{attribute 'GeneratedUsingTerminal: EK1122-0000-0018'}
{attribute addProperty BoxType "EK1122-0000-0018"}
{attribute addProperty Id "Beckhoff_CXxxxxsub_EK1100EK1100_AB5A94672A_0001_CX1100_0004_0000CX1100_AB5A94672A_0003_CX1100_0004_0002CX1100_AB5A94672A_0004_CX5010_EtherCAT_slaveCX5010_EtherCAT_slave_08881C8E20A_0005_CX5010_EtherCAT_slaveCX5010_EtherCAT_slave_08881C8E20A_0006_CX5020_EtherCAT_slaveCX5020_EtherCAT_slave_08881C8E20A_0007_CX5020_EtherCAT_slaveCX5020_EtherCAT_slave_08881C8E20A_0008_CX8010_EtherCAT_slaveCX8010_EtherCAT_slave_08881C8E20A_0009_CX8010_EtherCAT_slaveCX8010_EtherCAT_slave_08881C8E20A_0010_CX8110_EtherCAT_slaveCX8110_EtherCAT_slave_08881C8E20A_0011_CX2020_EtherCAT_slaveCX2020_EtherCAT_slave_08881C8E20A_0012_CX2020_EtherCAT_slaveCX2020_EtherCAT_slave_08881C8E20A_0013_CX2020_EtherCAT_slaveCX2020_EtherCAT_slave_08881C8E20A_0014_CX2030_EtherCAT_slaveCX2030_EtherCAT_slave_08881C8E20A_0015_CX2030_EtherCAT_slaveCX2030_EtherCAT_slave_08881C8E20A_0016_CX2030_EtherCAT_slaveCX2030_EtherCAT_slave_08881C8E20A_0017_CX2033_EtherCAT_slaveCX2033_EtherCAT_slave_08881C8E20A_0018_CX2040_EtherCAT_slaveCX2040_EtherCAT_slave_08881C8E20A_0019_CX2040_EtherCAT_slaveCX2040_EtherCAT_slave_08881C8E20A_0020_CX2040_EtherCAT_slaveCX2040_EtherCAT_slave_08881C8E20A_0021_CX2042_EtherCAT_slaveCX2042_EtherCAT_slave_08881C8E20A_0022_CX2043_EtherCAT_slaveCX2043_EtherCAT_slave_08881C8E20A_0023_CX2062_EtherCAT_slaveCX2062_EtherCAT_slave_08881C8E20A_0024_CX2072_EtherCAT_slaveCX2072_EtherCAT_slave_08881C8E20A_0025_CX9020_EtherCAT_slaveCX9020_EtherCAT_slave_08881C8E20A_0026_CX9020_EtherCAT_slaveCX9020_EtherCAT_slave_08881C8E20A_0027_CX5120_EtherCAT_slaveCX5120_EtherCAT_slave_08881C8E20A_0028_CX5130_EtherCAT_slaveCX5130_EtherCAT_slave_08881C8E20A_0029_CX5140_EtherCAT_slaveCX5140_EtherCAT_slave_08881C8E20A_0030_CX5230_EtherCAT_slaveCX5230_EtherCAT_slave_08881C8E20A_0031_CX5240_EtherCAT_slaveCX5240_EtherCAT_slave_08881C8E20A_0002_CX1100_0004_0001CX1100_AB5A94672"}
{attribute addProperty CRC "3494610126"}
{attribute addProperty Size "568"}
TYPE Beckhoff_CXxxxxEK1122_D04B84CE EXTENDS EK1122_AB5A9467 :
STRUCT
	{attribute addProperty Name "Beckhoff_CXxxxxsub_EK1100"}
	{attribute addProperty PreviousPort "Beckhoff CXxxxxEK1122 : D"}
	Beckhoff_CXxxxxsub_EK1100 : EK1100_AB5A9467;
	{attribute addProperty Name "A_0001_CX1100_0004_0000"}
	{attribute addProperty PreviousPort "Beckhoff CXxxxxsub EK1100 : C"}
	A_0001_CX1100_0004_0000 : CX1100_AB5A9467;
	{attribute addProperty Name "A_0003_CX1100_0004_0002"}
	{attribute addProperty PreviousPort "A_0001(CX1100-0004-0000) : C"}
	A_0003_CX1100_0004_0002 : CX1100_AB5A9467;
	{attribute addProperty Name "A_0004_CX5010_EtherCAT_slave"}
	{attribute addProperty PreviousPort "Beckhoff CXxxxxEK1122 : B"}
	A_0004_CX5010_EtherCAT_slave : CX5010_EtherCAT_slave_08881C8E;
	{attribute addProperty Name "A_0005_CX5010_EtherCAT_slave"}
	{attribute addProperty PreviousPort "A_0004 (CX5010 EtherCAT slave) : B"}
	A_0005_CX5010_EtherCAT_slave : CX5010_EtherCAT_slave_08881C8E;
	{attribute addProperty Name "A_0006_CX5020_EtherCAT_slave"}
	{attribute addProperty PreviousPort "A_0005 (CX5010 EtherCAT slave) : B"}
	A_0006_CX5020_EtherCAT_slave : CX5020_EtherCAT_slave_08881C8E;
	{attribute addProperty Name "A_0007_CX5020_EtherCAT_slave"}
	{attribute addProperty PreviousPort "A_0006 (CX5020 EtherCAT slave) : B"}
	A_0007_CX5020_EtherCAT_slave : CX5020_EtherCAT_slave_08881C8E;
	{attribute addProperty Name "A_0008_CX8010_EtherCAT_slave"}
	{attribute addProperty PreviousPort "A_0007 (CX5020 EtherCAT slave) : B"}
	A_0008_CX8010_EtherCAT_slave : CX8010_EtherCAT_slave_08881C8E;
	{attribute addProperty Name "A_0009_CX8010_EtherCAT_slave"}
	{attribute addProperty PreviousPort "A_0008 (CX8010 EtherCAT slave) : B"}
	A_0009_CX8010_EtherCAT_slave : CX8010_EtherCAT_slave_08881C8E;
	{attribute addProperty Name "A_0010_CX8110_EtherCAT_slave"}
	{attribute addProperty PreviousPort "A_0009 (CX8010 EtherCAT slave) : B"}
	A_0010_CX8110_EtherCAT_slave : CX8110_EtherCAT_slave_08881C8E;
	{attribute addProperty Name "A_0011_CX2020_EtherCAT_slave"}
	{attribute addProperty PreviousPort "A_0010 (CX8110 EtherCAT slave) : B"}
	A_0011_CX2020_EtherCAT_slave : CX2020_EtherCAT_slave_08881C8E;
	{attribute addProperty Name "A_0012_CX2020_EtherCAT_slave"}
	{attribute addProperty PreviousPort "A_0011 (CX2020 EtherCAT slave) : B"}
	A_0012_CX2020_EtherCAT_slave : CX2020_EtherCAT_slave_08881C8E;
	{attribute addProperty Name "A_0013_CX2020_EtherCAT_slave"}
	{attribute addProperty PreviousPort "A_0012 (CX2020 EtherCAT slave) : B"}
	A_0013_CX2020_EtherCAT_slave : CX2020_EtherCAT_slave_08881C8E;
	{attribute addProperty Name "A_0014_CX2030_EtherCAT_slave"}
	{attribute addProperty PreviousPort "A_0013 (CX2020 EtherCAT slave) : B"}
	A_0014_CX2030_EtherCAT_slave : CX2030_EtherCAT_slave_08881C8E;
	{attribute addProperty Name "A_0015_CX2030_EtherCAT_slave"}
	{attribute addProperty PreviousPort "A_0014 (CX2030 EtherCAT slave) : B"}
	A_0015_CX2030_EtherCAT_slave : CX2030_EtherCAT_slave_08881C8E;
	{attribute addProperty Name "A_0016_CX2030_EtherCAT_slave"}
	{attribute addProperty PreviousPort "A_0015 (CX2030 EtherCAT slave) : B"}
	A_0016_CX2030_EtherCAT_slave : CX2030_EtherCAT_slave_08881C8E;
	{attribute addProperty Name "A_0017_CX2033_EtherCAT_slave"}
	{attribute addProperty PreviousPort "A_0016 (CX2030 EtherCAT slave) : B"}
	A_0017_CX2033_EtherCAT_slave : CX2033_EtherCAT_slave_08881C8E;
	{attribute addProperty Name "A_0018_CX2040_EtherCAT_slave"}
	{attribute addProperty PreviousPort "A_0017 (CX2033 EtherCAT slave) : B"}
	A_0018_CX2040_EtherCAT_slave : CX2040_EtherCAT_slave_08881C8E;
	{attribute addProperty Name "A_0019_CX2040_EtherCAT_slave"}
	{attribute addProperty PreviousPort "A_0018 (CX2040 EtherCAT slave) : B"}
	A_0019_CX2040_EtherCAT_slave : CX2040_EtherCAT_slave_08881C8E;
	{attribute addProperty Name "A_0020_CX2040_EtherCAT_slave"}
	{attribute addProperty PreviousPort "A_0019 (CX2040 EtherCAT slave) : B"}
	A_0020_CX2040_EtherCAT_slave : CX2040_EtherCAT_slave_08881C8E;
	{attribute addProperty Name "A_0021_CX2042_EtherCAT_slave"}
	{attribute addProperty PreviousPort "A_0020 (CX2040 EtherCAT slave) : B"}
	A_0021_CX2042_EtherCAT_slave : CX2042_EtherCAT_slave_08881C8E;
	{attribute addProperty Name "A_0022_CX2043_EtherCAT_slave"}
	{attribute addProperty PreviousPort "A_0021 (CX2042 EtherCAT slave) : B"}
	A_0022_CX2043_EtherCAT_slave : CX2043_EtherCAT_slave_08881C8E;
	{attribute addProperty Name "A_0023_CX2062_EtherCAT_slave"}
	{attribute addProperty PreviousPort "A_0022 (CX2043 EtherCAT slave) : B"}
	A_0023_CX2062_EtherCAT_slave : CX2062_EtherCAT_slave_08881C8E;
	{attribute addProperty Name "A_0024_CX2072_EtherCAT_slave"}
	{attribute addProperty PreviousPort "A_0023 (CX2062 EtherCAT slave) : B"}
	A_0024_CX2072_EtherCAT_slave : CX2072_EtherCAT_slave_08881C8E;
	{attribute addProperty Name "A_0025_CX9020_EtherCAT_slave"}
	{attribute addProperty PreviousPort "A_0024 (CX2072 EtherCAT slave) : B"}
	A_0025_CX9020_EtherCAT_slave : CX9020_EtherCAT_slave_08881C8E;
	{attribute addProperty Name "A_0026_CX9020_EtherCAT_slave"}
	{attribute addProperty PreviousPort "A_0025 (CX9020 EtherCAT slave) : B"}
	A_0026_CX9020_EtherCAT_slave : CX9020_EtherCAT_slave_08881C8E;
	{attribute addProperty Name "A_0027_CX5120_EtherCAT_slave"}
	{attribute addProperty PreviousPort "A_0026 (CX9020 EtherCAT slave) : B"}
	A_0027_CX5120_EtherCAT_slave : CX5120_EtherCAT_slave_08881C8E;
	{attribute addProperty Name "A_0028_CX5130_EtherCAT_slave"}
	{attribute addProperty PreviousPort "A_0027 (CX5120 EtherCAT slave) : B"}
	A_0028_CX5130_EtherCAT_slave : CX5130_EtherCAT_slave_08881C8E;
	{attribute addProperty Name "A_0029_CX5140_EtherCAT_slave"}
	{attribute addProperty PreviousPort "A_0028 (CX5130 EtherCAT slave) : B"}
	A_0029_CX5140_EtherCAT_slave : CX5140_EtherCAT_slave_08881C8E;
	{attribute addProperty Name "A_0030_CX5230_EtherCAT_slave"}
	{attribute addProperty PreviousPort "A_0029 (CX5140 EtherCAT slave) : B"}
	A_0030_CX5230_EtherCAT_slave : CX5230_EtherCAT_slave_08881C8E;
	{attribute addProperty Name "A_0031_CX5240_EtherCAT_slave"}
	{attribute addProperty PreviousPort "A_0030 (CX5230 EtherCAT slave) : B"}
	A_0031_CX5240_EtherCAT_slave : CX5240_EtherCAT_slave_08881C8E;
	{attribute addProperty Name "A_0002_CX1100_0004_0001"}
	{attribute addProperty PreviousPort "A_0031 (CX5240 EtherCAT slave) : B"}
	A_0002_CX1100_0004_0001 : CX1100_AB5A9467;
END_STRUCT
END_TYPE

(* stored: Version 1.2.0.0, ProductVersion 3.1.4024.9
   DUT Beckhoff_CXxxxxEK1122_D04B84CE: Id {e77e590e-9a1a-47f2-b67b-cbc6bb363d27} *)
